FUNCTION_BLOCK CmdMetalSaltDosing (* Basic Function Block Type *)
  (* Standard: 61499-2 *)
  (* Version 0.0, 7/31/2024, Administrator, Schneider Electric, Template *)
  PACKAGE SE.Nereda;
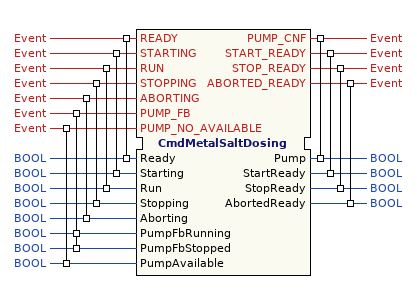
  EVENT_INPUT
    READY WITH Ready;
    STARTING WITH Starting;
    RUN WITH Run; (* Normal Execution Request *)
    STOPPING WITH Stopping;
    ABORTING WITH Aborting;
    PUMP_FB WITH PumpFbRunning, PumpFbStopped;
    PUMP_NO_AVAILABLE WITH PumpAvailable;
  END_EVENT
  EVENT_OUTPUT
    PUMP_CNF WITH Pump;
    START_READY WITH StartReady;
    STOP_READY WITH StopReady;
    ABORTED_READY WITH AbortedReady;
  END_EVENT
  VAR_INPUT
    Ready : BOOL;
    Starting : BOOL;
    Run : BOOL; (* Input event qualifier *)
    Stopping : BOOL;
    Aborting : BOOL;
    PumpFbRunning : BOOL;
    PumpFbStopped : BOOL;
    PumpAvailable : BOOL;
  END_VAR
  VAR_OUTPUT
    Pump : BOOL;
    StartReady : BOOL;
    StopReady : BOOL;
    AbortedReady : BOOL;
  END_VAR
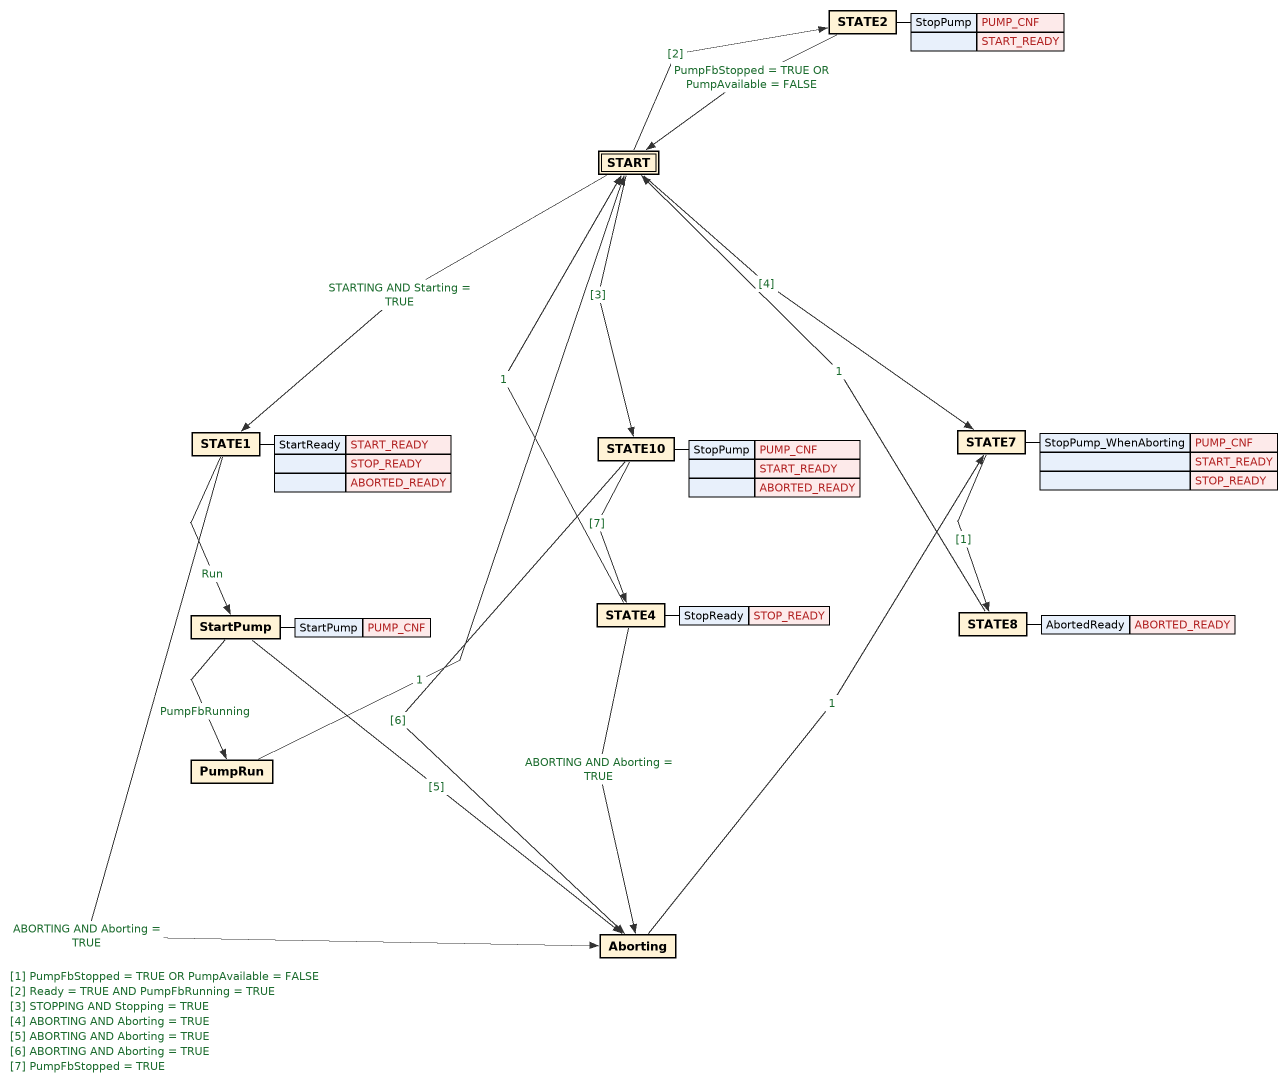
  EC_STATES
    START; (* Initial State *)
    STATE1 : StartReady -> START_READY, -> STOP_READY, -> ABORTED_READY; (* Normal execution *)
    StartPump : StartPump -> PUMP_CNF;
    STATE4 : StopReady -> STOP_READY;
    STATE8 : AbortedReady -> ABORTED_READY;
    Aborting;
    STATE2 : StopPump -> PUMP_CNF, -> START_READY;
    STATE7 : StopPump_WhenAborting -> PUMP_CNF, -> START_READY, -> STOP_READY;
    STATE10 : StopPump -> PUMP_CNF, -> START_READY, -> ABORTED_READY;
    PumpRun;
  END_STATES
  EC_TRANSITIONS
    START TO STATE1 := STARTING AND Starting = TRUE;
    STATE1 TO StartPump := Run;
    PumpRun TO START := 1;
    START TO STATE10 := STOPPING AND Stopping = TRUE;
    STATE4 TO START := 1;
    START TO STATE7 := ABORTING AND Aborting = TRUE;
    STATE8 TO START := 1;
    STATE1 TO Aborting := ABORTING AND Aborting = TRUE;
    Aborting TO STATE7 := 1;
    STATE4 TO Aborting := ABORTING AND Aborting = TRUE;
    START TO STATE2 := Ready = TRUE AND PumpFbRunning = TRUE;
    StartPump TO Aborting := ABORTING AND Aborting = TRUE;
    STATE7 TO STATE8 := PumpFbStopped = TRUE OR PumpAvailable = FALSE;
    STATE10 TO STATE4 := PumpFbStopped = TRUE;
    STATE2 TO START := PumpFbStopped = TRUE OR PumpAvailable = FALSE;
    STATE10 TO Aborting := ABORTING AND Aborting = TRUE;
    StartPump TO PumpRun := PumpFbRunning;
  END_TRANSITIONS
  ALGORITHM StartReady IN ST:
;
StartReady := TRUE;
StopReady := FALSE;
AbortedReady := FALSE;
  END_ALGORITHM
  ALGORITHM StopReady IN ST:
;
StopReady := TRUE;
  END_ALGORITHM
  ALGORITHM AbortedReady IN ST:
;
AbortedReady := TRUE;
  END_ALGORITHM
  ALGORITHM StartPump IN ST:
;
Pump := TRUE;
  END_ALGORITHM
  ALGORITHM StopPump IN ST:
;
Pump := FALSE;
StartReady := FALSE;
AbortedReady  := FALSE;
  END_ALGORITHM
  ALGORITHM StopPump_WhenAborting IN ST:
;
Pump := FALSE;
StartReady := FALSE;
StopReady := FALSE;
  END_ALGORITHM
END_FUNCTION_BLOCK
